//{{V2}}
ORGANIZATION_BLOCK OB1
TITLE= "Zyklisches Hauptprogramm"


AUTHOR:nb
FAMILY:nb
NAME:nb
VERSION:1.0


VAR_TEMP
       OB1_EV_CLASS:BYTE //Bits 0-3 = 1 (Coming event), Bits 4-7 = 1 (Event class 1)
       OB1_SCAN_1:BYTE //1 (Cold restart scan 1 of OB 1), 3 (Scan 2-n of OB 1)
       OB1_PRIORITY:BYTE //1 (Priority of 1 is lowest)
       OB1_OB_NUMBR:BYTE //1 (Organization block 1, OB1)
       OB1_RESERVED_1:BYTE //Reserved for system
       OB1_RESERVED_2:BYTE //Reserved for system
       OB1_PREV_CYCLE:INT //Cycle time of previous OB1 scan (milliseconds)
       OB1_MIN_CYCLE:INT //Minimum cycle time of OB1 (milliseconds)
       OB1_MAX_CYCLE:INT //Maximum cycle time of OB1 (milliseconds)
       OB1_DATE_TIME:DATE_AND_TIME //Date and time OB1 started
END_VAR
BEGIN

NETWORK
TITLE=
//{{a}}
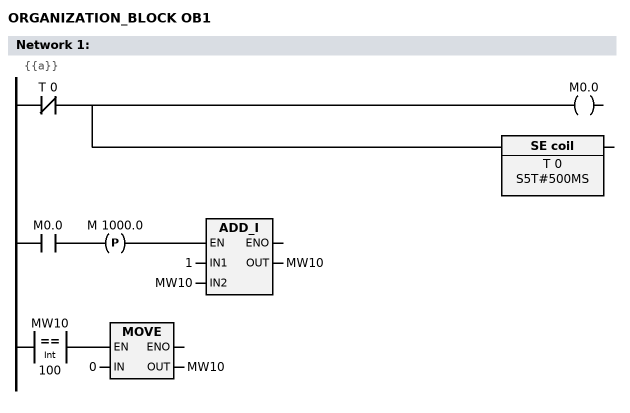

///////////
//Counter//
///////////

//Timer
       UN   T         0
       =    M0.0
       L    S5T#500MS
       SV   T         0

//Increment
       U    M0.0
       FP   M      1000.0
       SPBN _add
       L    1
       L    MW10
       +I
       T    MW10
_add:  NOP  0


//Reset
       L    MW10
       L    100
       ==I
       SPBN _res
       L    0
       T    MW10
_res:  NOP  0
NETWORK
TITLE=
//{{a}}

//EinerPos
       L    MW10
       L    10
       MOD
       T    MW14

//ZehnerPos
       L    MW10
       L    10
       /I
       T    MW12

//Concat
       L    MW12
       SLW            4
       L    MW14
       OW
       T    MW16

//Output
       L    MW16
       T    AW       10
END_ORGANIZATION_BLOCK
